// =========================================================
// 0. SYSTEM SAFE (oba NC stop prekidača moraju biti OK)
// =========================================================
bSystemSafe := GVL_IO.DI_Stop_Port AND GVL_IO.DI_Stop_Stbd;

// =========================================================
// 1. POZIV FUNKCIJSKIH BLOKOVA ZA VINČEVE
// =========================================================

// WINCH 1
fbWinch1(
    bIn_SafetyEnable := bSystemSafe,
    bBtn_Phy_Dir1    := GVL_IO.bBtn_Winch1_A,
    bBtn_Phy_Dir2    := GVL_IO.bBtn_Winch1_B,
    stHMI            := stWinch1_HMI,
    bValve_Dir1      => GVL_IO.bValve_Winch1_A,
    bValve_Dir2      => GVL_IO.bValve_Winch1_B
);

// WINCH 2
fbWinch2(
    bIn_SafetyEnable := bSystemSafe,
    bBtn_Phy_Dir1    := GVL_IO.bBtn_Winch2_A,
    bBtn_Phy_Dir2    := GVL_IO.bBtn_Winch2_B,
    stHMI            := stWinch2_HMI,
    bValve_Dir1      => GVL_IO.bValve_Winch2_A,
    bValve_Dir2      => GVL_IO.bValve_Winch2_B
);

// WINCH 3
fbWinch3(
    bIn_SafetyEnable := bSystemSafe,
    bBtn_Phy_Dir1    := GVL_IO.bBtn_Winch3_A,
    bBtn_Phy_Dir2    := GVL_IO.bBtn_Winch3_B,
    stHMI            := stWinch3_HMI,
    bValve_Dir1      => GVL_IO.bValve_Winch3_A,
    bValve_Dir2      => GVL_IO.bValve_Winch3_B
);

// =========================================================
// 2. DETEKCIJA OPTEREĆENJA (Koliko vinčeva radi?)
// =========================================================
iActiveCount := 0;

// Sada gledamo čisti izlaz iz FB-a koji već u sebi ima interlock i logiku!
IF fbWinch1.bReq_Pump THEN iActiveCount := iActiveCount + 1; END_IF
IF fbWinch2.bReq_Pump THEN iActiveCount := iActiveCount + 1; END_IF
IF fbWinch3.bReq_Pump THEN iActiveCount := iActiveCount + 1; END_IF

// Zastavica: Radi li itko?
GVL_IO.bAnyWinchActive := (iActiveCount > 0);

// =========================================================
// 3. UPRAVLJANJE RPM-om MOTORA (BOOST)
// =========================================================
bEngineIsOn := (GVL_IO.fEngineRPM_Scaled > 500.0);

IF GVL_IO.bAnyWinchActive AND bEngineIsOn THEN
    // Formula: Bazni ler + (BrojVinčeva * 200)
    GVL_IO.iRpmReq_Winches := iBaseRpm + (iActiveCount * iRpmPerWinch);
    
    // Sigurnosni limit RPM-a
    IF GVL_IO.iRpmReq_Winches > 2000 THEN 
        GVL_IO.iRpmReq_Winches := 2000; 
    END_IF
ELSE
    // Ako vinčevi ne rade ili motor stoji
    GVL_IO.iRpmReq_Winches := 0; 
END_IF

// =========================================================
// 4. LOGIKA DC PUMPE (BACKUP S OFF-DELAY TIMEMEROM)
// =========================================================

// Ako netko stišće vinč, a glavni motor ne vrti
// TOF (Timer Off) se pali momentalno, a gasi tek 5 sekundi nakon što pustiš tipku
tmrDCPumpOff(
    IN := (GVL_IO.bAnyWinchActive AND NOT bEngineIsOn), 
    PT := T#5S
);

GVL_IO.bDcPump_Start := tmrDCPumpOff.Q;

END_PROGRAM

// ---- POUs/FBs/FB_WinchControl.TcPOU
FUNCTION_BLOCK FB_WinchControl
VAR_INPUT
    (* --- FIZIČKI ULAZI --- *)
	bIn_SafetyEnable : BOOL;
    bBtn_Phy_Dir1    : BOOL; (* Fizička tipka (npr. nožni prekidač Slow) *)
    bBtn_Phy_Dir2    : BOOL; (* Fizička tipka (npr. nožni prekidač Fast) *)
END_VAR
VAR_OUTPUT
    (* --- FIZIČKI IZLAZI --- *)
    bValve_Dir1      : BOOL; 
    bValve_Dir2      : BOOL; 
    bReq_Pump        : BOOL; 
END_VAR
VAR_IN_OUT
    (* --- HMI PODACI --- *)
    stHMI            : ST_UcWinchControl;
END_VAR
VAR
    xCmd_Dir1        : BOOL;
    xCmd_Dir2        : BOOL;
END_VAR

(* ========================================================== *)
(* 1. INPUT MIXER (HMI vs HARDVER)                            *)
(* ========================================================== *)
IF stHMI.bManualEnable THEN
    (* Manual Mode: Slušamo samo HMI *)
    xCmd_Dir1 := stHMI.bBtn_Dir1;
    xCmd_Dir2 := stHMI.bBtn_Dir2;
ELSE
    (* Local Mode: Slušamo samo fizičke tipke *)
    xCmd_Dir1 := bBtn_Phy_Dir1;
    xCmd_Dir2 := bBtn_Phy_Dir2;
END_IF;

(* ========================================================== *)
(* 2. LOGIKA VITLA (Interlock + Pumpa)                        *)
(* ========================================================== *)
IF bIn_SafetyEnable AND NOT stHMI.bDisable THEN
    
    // Interlock: Ne može obje brzine/smjera odjednom
    IF xCmd_Dir1 AND xCmd_Dir2 THEN
        bValve_Dir1 := FALSE;
        bValve_Dir2 := FALSE;
        bReq_Pump   := FALSE;

    // Smjer 1 (npr. Slow / In)
    ELSIF xCmd_Dir1 THEN
        bValve_Dir1 := TRUE;
        bValve_Dir2 := FALSE;
        bReq_Pump   := TRUE; (* PUMPA ON *)

    // Smjer 2 (npr. Fast / Out)
    ELSIF xCmd_Dir2 THEN
        bValve_Dir1 := FALSE;
        bValve_Dir2 := TRUE;
        bReq_Pump   := TRUE; (* PUMPA ON *)
    
    // Mirovanje
    ELSE
        bValve_Dir1 := FALSE;
        bValve_Dir2 := FALSE;
        bReq_Pump   := FALSE;
    END_IF

ELSE
    // SAFETY STOP
    bValve_Dir1 := FALSE;
    bValve_Dir2 := FALSE;
    bReq_Pump   := FALSE;
END_IF

(* ========================================================== *)
(* 3. HMI FEEDBACK (Update strukture)                         *)
(* ========================================================== *)
stHMI.bValve_Dir1     := bValve_Dir1;
stHMI.bValve_Dir2     := bValve_Dir2;
stHMI.bReq_Pump       := bReq_Pump;

stHMI.bSts_SystemSafe := bIn_SafetyEnable AND NOT stHMI.bDisable;
stHMI.bSts_ManualEn   := stHMI.bManualEnable;

END_FUNCTION_BLOCK

// ---- POUs/Sim/PRG_SimDoors.TcPOU
PROGRAM PRG_SimDoors
VAR
    (* Parametri za VRATA *)
    fRiseSpeed   : REAL := 0.04; 
    fDropSpeed   : REAL := 0.001; 
    fTankSpeed   : REAL := 2.0;  
    
    (* Tajmeri za simulaciju kretanja VENTILA *)
    tonP1, tonP2, tonP3 : TON;
    tonS1, tonS2, tonS3 : TON;
    tonTunel           : TON;
    
    tValveTime : TIME := T#1.5S; (* Brže od 3s timeouta u FB-u! *)
    bSimActive : BOOL := TRUE;
	
	// Timer koji simulira koliko dugo ima vode u cijevima nakon paljenja pumpe
	tmrVodaTrajanje : TON;
    tVrijemeRada    : TIME := T#10S; // Koliko dugo ima vode u tanku
    bTankPrazan     : BOOL;         // Zasun koji sprječava titranjeEND_VAR
END_VAR

// -----------------------------------------------------------
// 0. GLAVNI PREKIDAČ SIMULATORA
// -----------------------------------------------------------
IF NOT bSimActive THEN
    RETURN;
END_IF

// -----------------------------------------------------------
// 1. SIMULACIJA VRATA (FWD & AFT)
// -----------------------------------------------------------

// --- FWD VRATA ---
IF GVL_IO.DO_DoorFwd_Open THEN
    GVL_IO.fPressure_FWD_A := GVL_IO.fPressure_FWD_A + fRiseSpeed;
    GVL_IO.fPressure_FWD_B := GVL_IO.fPressure_FWD_B - fTankSpeed;
ELSIF GVL_IO.DO_DoorFwd_Close THEN
    GVL_IO.fPressure_FWD_B := GVL_IO.fPressure_FWD_B + fRiseSpeed;
    GVL_IO.fPressure_FWD_A := GVL_IO.fPressure_FWD_A - fTankSpeed;
ELSE
    GVL_IO.fPressure_FWD_A := GVL_IO.fPressure_FWD_A - fDropSpeed;
    GVL_IO.fPressure_FWD_B := GVL_IO.fPressure_FWD_B - fDropSpeed;
END_IF

// --- AFT VRATA ---
IF GVL_IO.DO_DoorAft_Open THEN
    GVL_IO.fPressure_AFT_A := GVL_IO.fPressure_AFT_A + fRiseSpeed;
    GVL_IO.fPressure_AFT_B := GVL_IO.fPressure_AFT_B - fTankSpeed;
ELSIF GVL_IO.DO_DoorAft_Close THEN
    GVL_IO.fPressure_AFT_B := GVL_IO.fPressure_AFT_B + fRiseSpeed;
    GVL_IO.fPressure_AFT_A := GVL_IO.fPressure_AFT_A - fTankSpeed;
ELSE
    GVL_IO.fPressure_AFT_A := GVL_IO.fPressure_AFT_A - fDropSpeed;
    GVL_IO.fPressure_AFT_B := GVL_IO.fPressure_AFT_B - fDropSpeed;
END_IF

// Ograničenja tlaka (da ne ide u minus ili beskonačno)
GVL_IO.fPressure_FWD_A := LIMIT(0.0, GVL_IO.fPressure_FWD_A, 150.0);
GVL_IO.fPressure_FWD_B := LIMIT(0.0, GVL_IO.fPressure_FWD_B, 150.0);
GVL_IO.fPressure_AFT_A := LIMIT(0.0, GVL_IO.fPressure_AFT_A, 150.0);
GVL_IO.fPressure_AFT_B := LIMIT(0.0, GVL_IO.fPressure_AFT_B, 150.0);

// -----------------------------------------------------------
// 2. SIMULACIJA BALAST VENTILA (Feedback)
// -----------------------------------------------------------

// PORT 1
tonP1(IN := GVL_IO.DO_BAL_P1, PT := tValveTime);
IF GVL_IO.DO_BAL_P1 THEN
    GVL_IO.DI_BAL_P1_OPEN_FB  := tonP1.Q;
    GVL_IO.DI_BAL_P1_CLOSE_FB := FALSE;
ELSE
    GVL_IO.DI_BAL_P1_OPEN_FB  := FALSE;
    GVL_IO.DI_BAL_P1_CLOSE_FB := TRUE;
END_IF

// PORT 2
tonP2(IN := GVL_IO.DO_BAL_P2, PT := tValveTime);
IF GVL_IO.DO_BAL_P2 THEN
    GVL_IO.DI_BAL_P2_OPEN_FB  := tonP2.Q;
    GVL_IO.DI_BAL_P2_CLOSE_FB := FALSE;
ELSE
    GVL_IO.DI_BAL_P2_OPEN_FB  := FALSE;
    GVL_IO.DI_BAL_P2_CLOSE_FB := TRUE;
END_IF

// PORT 3
tonP3(IN := GVL_IO.DO_BAL_P3, PT := tValveTime);
IF GVL_IO.DO_BAL_P3 THEN
    GVL_IO.DI_BAL_P3_OPEN_FB  := tonP3.Q;
    GVL_IO.DI_BAL_P3_CLOSE_FB := FALSE;
ELSE
    GVL_IO.DI_BAL_P3_OPEN_FB  := FALSE;
    GVL_IO.DI_BAL_P3_CLOSE_FB := TRUE;
END_IF

// STBD 1
tonS1(IN := GVL_IO.DO_BAL_S1, PT := tValveTime);
IF GVL_IO.DO_BAL_S1 THEN
    GVL_IO.DI_BAL_S1_OPEN_FB  := tonS1.Q;
    GVL_IO.DI_BAL_S1_CLOSE_FB := FALSE;
ELSE
    GVL_IO.DI_BAL_S1_OPEN_FB  := FALSE;
    GVL_IO.DI_BAL_S1_CLOSE_FB := TRUE;
END_IF

// STBD 2
tonS2(IN := GVL_IO.DO_BAL_S2, PT := tValveTime);
IF GVL_IO.DO_BAL_S2 THEN
    GVL_IO.DI_BAL_S2_OPEN_FB  := tonS2.Q;
    GVL_IO.DI_BAL_S2_CLOSE_FB := FALSE;
ELSE
    GVL_IO.DI_BAL_S2_OPEN_FB  := FALSE;
    GVL_IO.DI_BAL_S2_CLOSE_FB := TRUE;
END_IF

// STBD 3
tonS3(IN := GVL_IO.DO_BAL_S3, PT := tValveTime);
IF GVL_IO.DO_BAL_S3 THEN
    GVL_IO.DI_BAL_S3_OPEN_FB  := tonS3.Q;
    GVL_IO.DI_BAL_S3_CLOSE_FB := FALSE;
ELSE
    GVL_IO.DI_BAL_S3_OPEN_FB  := FALSE;
    GVL_IO.DI_BAL_S3_CLOSE_FB := TRUE;
END_IF

// -----------------------------------------------------------
// 3. SIMULACIJA TUNEL PUMP VENTILA
// -----------------------------------------------------------
tonTunel(IN := GVL_IO.DO_TUNEL_VALVE, PT := tValveTime);
IF GVL_IO.DO_TUNEL_VALVE THEN
    GVL_IO.DI_TUNEL_OPEN_FB  := tonTunel.Q;
    GVL_IO.DI_TUNEL_CLOSE_FB := FALSE;
ELSE
    GVL_IO.DI_TUNEL_OPEN_FB  := FALSE;
    GVL_IO.DI_TUNEL_CLOSE_FB := TRUE;
END_IF

// ==========================================================
// 4. SIMULACIJA SONDI S TIMEROM (NESTANAK VODE)
// ==========================================================

// --- SIMULACIJA NESTANKA VODE ---
// Timer mjeri koliko dugo pumpa (Clutch) vrti
tmrVodaTrajanje(IN := GVL_IO.DO_TunelClutch, PT := tVrijemeRada);

// Kad timer odradi, "ispraznili" smo tank
IF tmrVodaTrajanje.Q THEN
    bTankPrazan := TRUE; 
END_IF

// Resetiramo tank tek kad se ugasi komanda pumpe (da možemo opet testirati)
IF NOT GVL_HMI.bCmdRun_TunelPump THEN
    bTankPrazan := FALSE;
END_IF

// --- LOGIKA SONDI ---
IF GVL_IO.DO_SondePower THEN
    // Port Sonda: ima struje, ventil je na Portu I tank NIJE prazan
    GVL_IO.DI_Sonda_Port := GVL_IO.DI_TUNEL_OPEN_FB AND NOT bTankPrazan;
    
    // Stbd Sonda: ima struje, ventil je na Stbd I tank NIJE prazan
    GVL_IO.DI_Sonda_Stbd := GVL_IO.DI_TUNEL_CLOSE_FB AND NOT bTankPrazan;
ELSE
    GVL_IO.DI_Sonda_Port := FALSE;
    GVL_IO.DI_Sonda_Stbd := FALSE;
END_IF

END_PROGRAM

// ---- POUs/PRG_HmiLeds.TcPOU
PROGRAM PRG_HmiLeds
VAR
END_VAR


// ============================================================
// HMI LED STATUSI
// Cyan=Otvoren, Green=Zatvoren, Orange(Yellow)=Putuje, Red=Greška
// ============================================================

// --- MOTOR ---
GVL_HMI.bLed_Engine_Green := GVL_ENGINE.bEngineRunning;

// --- PUMPA ---
GVL_HMI.bLed_Pump_Cyan := GVL_HMI.bCmdRun_TunelPump;
GVL_HMI.bLed_Pump_Red  := FALSE;

// --- PORT VENTILI ---
// P1
IF GVL_HMI.bAlarm_P1 THEN
    GVL_HMI.bLed_P1_Red := TRUE;  GVL_HMI.bLed_P1_Cyan := FALSE; GVL_HMI.bLed_P1_Yellow := FALSE; GVL_HMI.bLed_P1_Green := FALSE;
ELSIF GVL_HMI.eState_P1 = E_ValveState.VALVE_OPEN THEN
    GVL_HMI.bLed_P1_Red := FALSE; GVL_HMI.bLed_P1_Cyan := TRUE;  GVL_HMI.bLed_P1_Yellow := FALSE; GVL_HMI.bLed_P1_Green := FALSE;
ELSIF GVL_HMI.eState_P1 = E_ValveState.VALVE_UNKNOWN THEN
    GVL_HMI.bLed_P1_Red := FALSE; GVL_HMI.bLed_P1_Cyan := FALSE; GVL_HMI.bLed_P1_Yellow := TRUE;  GVL_HMI.bLed_P1_Green := FALSE;
ELSE // VALVE_CLOSED
    GVL_HMI.bLed_P1_Red := FALSE; GVL_HMI.bLed_P1_Cyan := FALSE; GVL_HMI.bLed_P1_Yellow := FALSE; GVL_HMI.bLed_P1_Green := TRUE;
END_IF

// P2
IF GVL_HMI.bAlarm_P2 THEN
    GVL_HMI.bLed_P2_Red := TRUE;  GVL_HMI.bLed_P2_Cyan := FALSE; GVL_HMI.bLed_P2_Yellow := FALSE; GVL_HMI.bLed_P2_Green := FALSE;
ELSIF GVL_HMI.eState_P2 = E_ValveState.VALVE_OPEN THEN
    GVL_HMI.bLed_P2_Red := FALSE; GVL_HMI.bLed_P2_Cyan := TRUE;  GVL_HMI.bLed_P2_Yellow := FALSE; GVL_HMI.bLed_P2_Green := FALSE;
ELSIF GVL_HMI.eState_P2 = E_ValveState.VALVE_UNKNOWN THEN
    GVL_HMI.bLed_P2_Red := FALSE; GVL_HMI.bLed_P2_Cyan := FALSE; GVL_HMI.bLed_P2_Yellow := TRUE;  GVL_HMI.bLed_P2_Green := FALSE;
ELSE
    GVL_HMI.bLed_P2_Red := FALSE; GVL_HMI.bLed_P2_Cyan := FALSE; GVL_HMI.bLed_P2_Yellow := FALSE; GVL_HMI.bLed_P2_Green := TRUE;
END_IF

// P3
IF GVL_HMI.bAlarm_P3 THEN
    GVL_HMI.bLed_P3_Red := TRUE;  GVL_HMI.bLed_P3_Cyan := FALSE; GVL_HMI.bLed_P3_Yellow := FALSE; GVL_HMI.bLed_P3_Green := FALSE;
ELSIF GVL_HMI.eState_P3 = E_ValveState.VALVE_OPEN THEN
    GVL_HMI.bLed_P3_Red := FALSE; GVL_HMI.bLed_P3_Cyan := TRUE;  GVL_HMI.bLed_P3_Yellow := FALSE; GVL_HMI.bLed_P3_Green := FALSE;
ELSIF GVL_HMI.eState_P3 = E_ValveState.VALVE_UNKNOWN THEN
    GVL_HMI.bLed_P3_Red := FALSE; GVL_HMI.bLed_P3_Cyan := FALSE; GVL_HMI.bLed_P3_Yellow := TRUE;  GVL_HMI.bLed_P3_Green := FALSE;
ELSE
    GVL_HMI.bLed_P3_Red := FALSE; GVL_HMI.bLed_P3_Cyan := FALSE; GVL_HMI.bLed_P3_Yellow := FALSE; GVL_HMI.bLed_P3_Green := TRUE;
END_IF

// --- STBD VENTILI ---
// S1
IF GVL_HMI.bAlarm_S1 THEN
    GVL_HMI.bLed_S1_Red := TRUE;  GVL_HMI.bLed_S1_Cyan := FALSE; GVL_HMI.bLed_S1_Yellow := FALSE; GVL_HMI.bLed_S1_Green := FALSE;
ELSIF GVL_HMI.eState_S1 = E_ValveState.VALVE_OPEN THEN
    GVL_HMI.bLed_S1_Red := FALSE; GVL_HMI.bLed_S1_Cyan := TRUE;  GVL_HMI.bLed_S1_Yellow := FALSE; GVL_HMI.bLed_S1_Green := FALSE;
ELSIF GVL_HMI.eState_S1 = E_ValveState.VALVE_UNKNOWN THEN
    GVL_HMI.bLed_S1_Red := FALSE; GVL_HMI.bLed_S1_Cyan := FALSE; GVL_HMI.bLed_S1_Yellow := TRUE;  GVL_HMI.bLed_S1_Green := FALSE;
ELSE
    GVL_HMI.bLed_S1_Red := FALSE; GVL_HMI.bLed_S1_Cyan := FALSE; GVL_HMI.bLed_S1_Yellow := FALSE; GVL_HMI.bLed_S1_Green := TRUE;
END_IF

// S2
IF GVL_HMI.bAlarm_S2 THEN
    GVL_HMI.bLed_S2_Red := TRUE;  GVL_HMI.bLed_S2_Cyan := FALSE; GVL_HMI.bLed_S2_Yellow := FALSE; GVL_HMI.bLed_S2_Green := FALSE;
ELSIF GVL_HMI.eState_S2 = E_ValveState.VALVE_OPEN THEN
    GVL_HMI.bLed_S2_Red := FALSE; GVL_HMI.bLed_S2_Cyan := TRUE;  GVL_HMI.bLed_S2_Yellow := FALSE; GVL_HMI.bLed_S2_Green := FALSE;
ELSIF GVL_HMI.eState_S2 = E_ValveState.VALVE_UNKNOWN THEN
    GVL_HMI.bLed_S2_Red := FALSE; GVL_HMI.bLed_S2_Cyan := FALSE; GVL_HMI.bLed_S2_Yellow := TRUE;  GVL_HMI.bLed_S2_Green := FALSE;
ELSE
    GVL_HMI.bLed_S2_Red := FALSE; GVL_HMI.bLed_S2_Cyan := FALSE; GVL_HMI.bLed_S2_Yellow := FALSE; GVL_HMI.bLed_S2_Green := TRUE;
END_IF

// S3
IF GVL_HMI.bAlarm_S3 THEN
    GVL_HMI.bLed_S3_Red := TRUE;  GVL_HMI.bLed_S3_Cyan := FALSE; GVL_HMI.bLed_S3_Yellow := FALSE; GVL_HMI.bLed_S3_Green := FALSE;
ELSIF GVL_HMI.eState_S3 = E_ValveState.VALVE_OPEN THEN
    GVL_HMI.bLed_S3_Red := FALSE; GVL_HMI.bLed_S3_Cyan := TRUE;  GVL_HMI.bLed_S3_Yellow := FALSE; GVL_HMI.bLed_S3_Green := FALSE;
ELSIF GVL_HMI.eState_S3 = E_ValveState.VALVE_UNKNOWN THEN
    GVL_HMI.bLed_S3_Red := FALSE; GVL_HMI.bLed_S3_Cyan := FALSE; GVL_HMI.bLed_S3_Yellow := TRUE;  GVL_HMI.bLed_S3_Green := FALSE;
ELSE
    GVL_HMI.bLed_S3_Red := FALSE; GVL_HMI.bLed_S3_Cyan := FALSE; GVL_HMI.bLed_S3_Yellow := FALSE; GVL_HMI.bLed_S3_Green := TRUE;
END_IF

// --- TUNEL VENTIL ---
IF GVL_HMI.bAlarm_Tunel THEN
    GVL_HMI.bLed_Tunel_Red := TRUE;  GVL_HMI.bLed_Tunel_Cyan := FALSE; GVL_HMI.bLed_Tunel_Yellow := FALSE; GVL_HMI.bLed_Tunel_Green := FALSE;
ELSIF GVL_HMI.eState_Tunel = E_ValveState.VALVE_OPEN THEN
    GVL_HMI.bLed_Tunel_Red := FALSE; GVL_HMI.bLed_Tunel_Cyan := TRUE;  GVL_HMI.bLed_Tunel_Yellow := FALSE; GVL_HMI.bLed_Tunel_Green := FALSE;
ELSIF GVL_HMI.eState_Tunel = E_ValveState.VALVE_UNKNOWN THEN
    GVL_HMI.bLed_Tunel_Red := FALSE; GVL_HMI.bLed_Tunel_Cyan := FALSE; GVL_HMI.bLed_Tunel_Yellow := TRUE;  GVL_HMI.bLed_Tunel_Green := FALSE;
ELSE
    GVL_HMI.bLed_Tunel_Red := FALSE; GVL_HMI.bLed_Tunel_Cyan := FALSE; GVL_HMI.bLed_Tunel_Yellow := FALSE; GVL_HMI.bLed_Tunel_Green := TRUE;
END_IF

// --- VRATA FWD ---
IF GVL_HMI.bAlarm_DoorFwd THEN
    GVL_HMI.bLed_DoorFwd_Red := TRUE;  GVL_HMI.bLed_DoorFwd_Cyan := FALSE; GVL_HMI.bLed_DoorFwd_Yellow := FALSE; GVL_HMI.bLed_DoorFwd_Green := FALSE;
ELSIF GVL_HMI.eState_DoorFwd = 1 THEN // OPEN
    GVL_HMI.bLed_DoorFwd_Red := FALSE; GVL_HMI.bLed_DoorFwd_Cyan := TRUE;  GVL_HMI.bLed_DoorFwd_Yellow := FALSE; GVL_HMI.bLed_DoorFwd_Green := FALSE;
ELSIF GVL_HMI.eState_DoorFwd = 0 THEN // PUTUJE
    GVL_HMI.bLed_DoorFwd_Red := FALSE; GVL_HMI.bLed_DoorFwd_Cyan := FALSE; GVL_HMI.bLed_DoorFwd_Yellow := TRUE;  GVL_HMI.bLed_DoorFwd_Green := FALSE;
ELSE // CLOSED
    GVL_HMI.bLed_DoorFwd_Red := FALSE; GVL_HMI.bLed_DoorFwd_Cyan := FALSE; GVL_HMI.bLed_DoorFwd_Yellow := FALSE; GVL_HMI.bLed_DoorFwd_Green := TRUE;
END_IF

// --- VRATA AFT ---
IF GVL_HMI.bAlarm_DoorAft THEN
    GVL_HMI.bLed_DoorAft_Red := TRUE;  GVL_HMI.bLed_DoorAft_Cyan := FALSE; GVL_HMI.bLed_DoorAft_Yellow := FALSE; GVL_HMI.bLed_DoorAft_Green := FALSE;
ELSIF GVL_HMI.eState_DoorAft = 1 THEN // OPEN
    GVL_HMI.bLed_DoorAft_Red := FALSE; GVL_HMI.bLed_DoorAft_Cyan := TRUE;  GVL_HMI.bLed_DoorAft_Yellow := FALSE; GVL_HMI.bLed_DoorAft_Green := FALSE;
ELSIF GVL_HMI.eState_DoorAft = 0 THEN // PUTUJE
    GVL_HMI.bLed_DoorAft_Red := FALSE; GVL_HMI.bLed_DoorAft_Cyan := FALSE; GVL_HMI.bLed_DoorAft_Yellow := TRUE;  GVL_HMI.bLed_DoorAft_Green := FALSE;
ELSE // CLOSED
    GVL_HMI.bLed_DoorAft_Red := FALSE; GVL_HMI.bLed_DoorAft_Cyan := FALSE; GVL_HMI.bLed_DoorAft_Yellow := FALSE; GVL_HMI.bLed_DoorAft_Green := TRUE;
END_IF

END_PROGRAM

// ---- POUs/DirectMotorControl.TcPOU
PROGRAM DirectMotorControl
VAR
	bHMI_RESET: BOOL;	// reset gresaka
 
	bMotorOn: BOOL;
	rVelocitySetpoint: LREAL;
	rPotFeedback_V: REAL;
	rPotFeedback_Radno_Perc: LREAL;
	rRadno_Min_Pos: LREAL;	// Radni limit 0%
	rRadno_Max_Pos: REAL;	// Radni limit 100%
	
   // Realni Potenciometar - u RAW vrijednosti
    cPotMin: REAL := 0.55;             // kΩ ili V
    cPotMax: REAL := 7.16;             // kΩ ili V
	rLinearPosition: LREAL;	// realna pozicija max hoda od 81mm

	rLinearPosition_LimMin: LREAL;	// Limit iskljucenja
	rLinearPosition_LimMAx: LREAL;	// Limit iskljucenja
	
	// Parametri regulacije (NOVO)
    rSetpoint: REAL := 50.0;      // Željena pozicija 0-100%
    rMinVelocity: REAL := 10.0;     // Min brzina za start %
    rMaxVelocity: REAL := 100.0;   // Max brzina %
    rDeadband: REAL := 1.0;        // Deadband ±1%
    rKp: REAL := 10;              // P pojačanje
    
    // Procesne varijable (NOVO)
    rError: REAL;	// greska slijeđenja
    rVelocityCmd: REAL;
    bInDeadband: BOOL;	// Unutar pozicije
	
   // NOVO - Rampa varijable
    rSetpointTarget: REAL := 50.0;    // Ciljna pozicija
    rRampRate: REAL := 50.0;          // Brzina rampe [%/s]
	
   // NOVO - Računanje brzine
    rActualVelocity: REAL;        // Stvarna brzina [%/s]
    rActualVelocityRPM: REAL;     // Stvarna brzina [RPM]
    rLastPosition: LREAL;          // Prethodna pozicija
    rDeltaPosition: LREAL;         // Promjena pozicije
    fbVelocityTimer: TON;         // Timer za uzorkovanje
    tSampleTime: TIME := T#50MS;  // Vrijeme uzorkovanja
    
    // Filter za brzinu (opciono)
    rVelocityFiltered: REAL;
    rFilterConst: REAL := 0.3;    // Filter konstanta (0.1-0.5)

	rMotorVoltage: LREAL;
	rMotorCurrent: LREAL;
	Tgen1: TON;
	bTick: BOOL;
	TP1: TP;
	bTakt: BOOL;
	rSetpointTarget_Min: REAL:=0.0;
	rSetpointTarget_Max: REAL:=100.0;
	
	bSetVelOverPoz: BOOL;
	bSetVelOverNeg: BOOL;
	
	R_Tgen1: R_TRIG;

	Kn: REAL;
END_VAR

// Test postavke za reverziranje 0..100%
(*
Tgen1(IN:=NOT bTick , PT:=T#5S , Q=>bTick , ET=> );
TP1(IN:=bTick , PT:=Tgen1.PT/2 , Q=>bTakt , ET=> );
*)
Tgen1(IN:=bInDeadband , PT:=T#2S , Q=>bTick , ET=> );
R_Tgen1(CLK:=Tgen1.Q , Q=>bTick );
IF bTick THEN
	bTakt:=NOT bTakt;
END_IF

// MODIFICIRANO - postavljamo target umjesto direktnog setpointa
IF bTakt THEN
    rSetpointTarget := rSetpointTarget_Min;
ELSE
    rSetpointTarget := rSetpointTarget_Max;
END_IF

// NOVO - Rampiranje setpointa
IF rSetpoint < rSetpointTarget - 0.1 THEN
    // Rampiranje gore
    rSetpoint := rSetpoint + rRampRate * 0.01; // 0.01 = 10ms ciklus
    IF rSetpoint > rSetpointTarget THEN
        rSetpoint := rSetpointTarget;
    END_IF
ELSIF rSetpoint > rSetpointTarget + 0.1 THEN
    // Rampiranje dolje  
    rSetpoint := rSetpoint - rRampRate * 0.01;
    IF rSetpoint < rSetpointTarget THEN
        rSetpoint := rSetpointTarget;
    END_IF
END_IF


// Skaliranje 1 okretajng pot pozicije.
rPotFeedback_V:=10.0*iwPotFeedback/32767;	//napon na ulazu u EL3002
// pozicija pomaka = 81mm
rLinearPosition:=81.0*(rPotFeedback_V-cPotMin)/(cPotMax-cPotMin);
// Sigurnosni limiti + / - 
rLinearPosition_LimMin:=5.0;	// Safe limit negativan
rLinearPosition_LimMAx:=75.0;	// Safe limit pozitivan

// Sigurnosni limiti - iskljucuju Motor
IF (rLinearPosition < rLinearPosition_LimMin) OR  (rLinearPosition > rLinearPosition_LimMAx) THEN
	bMotorOn:=FALSE;
END_IF

// Radno podrucje pomaka 0..100% = MORA BITI UNUTAR SIGURNOSNIH LIMITA
rRadno_Min_Pos:=10.0;
rRadno_Max_Pos:=70.0;
rPotFeedback_Radno_Perc:= 100*(rLinearPosition-rRadno_Min_Pos)/(rRadno_Max_Pos-rRadno_Min_Pos);

// Open-loop kontrola
// Setpoint 0..100% = 0.....
// Limit za pretvorbu u integer 
// greska ako je veće od 32766 i manje od - 32766

// Kn ke multiplikator za setpoint u granicama -32000 .. 32000 / 0.100%
Kn:=320; // ako ide do napona napajanja 12V onda na 100% steka
// reset iz HMI
// bReset := FALSE;
IF bHMI_RESET THEN
	bSetVelOverPoz:=FALSE;
	bSetVelOverNeg:=FALSE;
    bReset := TRUE;
END_IF

IF NOT bError THEN
	bReset := FALSE;
END_IF


IF (rVelocitySetpoint*Kn > 32766) THEN
	bSetVelOverPoz:=TRUE;
END_IF
IF (rVelocitySetpoint*Kn < -32766) THEN
	bSetVelOverNeg:=TRUE;
END_IF
IF bSetVelOverPoz OR bSetVelOverNeg THEN
	bMotorOn:=FALSE;
ELSE
	nVelocitySetpoint:=LREAL_TO_INT(rVelocitySetpoint*Kn);
END_IF

// Dodano
// NOVO - POZICIJSKA REGULACIJA
IF bMotorOn THEN
    // Računaj grešku pozicije
    rError := rSetpoint - rPotFeedback_Radno_Perc;
    
    // Provjeri deadband
    bInDeadband := ABS(rError) <= rDeadband;
    
    IF NOT bInDeadband THEN
        // P regulator
        rVelocityCmd := rError * rKp;
        
        // Ograniči na max brzinu
        rVelocityCmd := LIMIT(-rMaxVelocity, rVelocityCmd, rMaxVelocity);
        
        // Primjeni minimalnu brzinu
        IF (ABS(rVelocityCmd) > 0.1) AND (ABS(rVelocityCmd) < rMinVelocity) THEN
            IF rVelocityCmd > 0 THEN
                rVelocityCmd := rMinVelocity;
            ELSE
                rVelocityCmd := -rMinVelocity;
            END_IF
        END_IF
    ELSE
        // Unutar deadband - zaustavi
        rVelocityCmd := 0.0;
    END_IF
    
    // Postavi brzinu
    rVelocitySetpoint := rVelocityCmd;
ELSE
    rVelocitySetpoint := 0.0;
END_IF

// Računanje brzine iz promjene pozicije

// Timer za periodičko računanje brzine
fbVelocityTimer(IN:= NOT fbVelocityTimer.Q, PT:= tSampleTime);

// Računaj brzinu kada timer istekne
IF fbVelocityTimer.Q THEN
    // Promjena pozicije u %
    rDeltaPosition := rLinearPosition - rLastPosition;
    
    // Brzina u mm/s !!!! NAVOJ IMA MULTIPLIKATOR X2
    rActualVelocity := rDeltaPosition / 0.05 / 2 ; // 50ms = 0.05s
    
    // Spremi trenutnu poziciju
    rLastPosition := rLinearPosition;
    
    // Filter brzine (PT1)
    rVelocityFiltered := rVelocityFiltered * (1.0 - rFilterConst) + 
                        rActualVelocity * rFilterConst;
END_IF

// Preračun u druge jedinice
// 81mm =  171.3 okr Motora
// RPM motora
rActualVelocityRPM := 60*171.3*rActualVelocity/81 ;


// =======================  DIVER PREMA TERMINALU

// driver prema EL7342
IF bMotorOn THEN
    bEnable := TRUE;
    bReduceTorque := FALSE;  // Puna snaga
 ELSE
    bEnable := FALSE;
    bReduceTorque := FALSE;
    nVelocitySetpoint := 0;
END_IF

(*
IF bMotorOn THEN
    nControlWord := 16#000F;
ELSE
    nControlWord := 16#0006;
    nVelocitySetpoint := 0;
END_IF
*)

rMotorVoltage:=(UINT_TO_INT(nMotorVoltage))/1000.0;
rMotorCurrent:=(UINT_TO_INT(nMotorCurrent))/1000.0;

END_PROGRAM

// ---- POUs/PRG_Sequence.TcPOU
PROGRAM PRG_Sequence
VAR
    eTargetMode  : E_SystemMode := 0;
    bTurbineSafe : BOOL;
    
    (* Nova varijabla: Netko treba vodu *)
    bWaterRequest : BOOL; 
	
	(* Triggeri za Tipku 4 s obje tipkovnice *)
    rtMode_ID10   : R_TRIG;
    rtMode_ID11   : R_TRIG;
END_VAR

// =========================================================
// 1. OBRADA ZAHTJEVA ZA MOD (Tipka 4)
// =========================================================

// Sigurnost: Ne mijenjaj mod ako turbina vrti prebrzo
bTurbineSafe := (GVL_IO.fEngineRPM_Scaled < 900.0); 

rtMode_ID10(CLK := GVL_CAN.ID10_Status[4]);
rtMode_ID11(CLK := GVL_CAN.ID11_Status[4]);

// Ako je sigurno, kružimo kroz modove pritiskom na Tipku 4
IF bTurbineSafe AND (rtMode_ID10.Q OR rtMode_ID11.Q) THEN
    CASE eTargetMode OF
        E_SystemMode.MODE_IDLE:  
            eTargetMode := E_SystemMode.MODE_DRIVE; // Prebaci na Drive (Zeleno)
            
        E_SystemMode.MODE_DRIVE: 
            eTargetMode := E_SystemMode.MODE_SAIL;  // Prebaci na Sail (Plavo)
            
        E_SystemMode.MODE_SAIL:  
            eTargetMode := E_SystemMode.MODE_IDLE;  // Vrati na Idle (Off)
    END_CASE
END_IF

// Zadržavamo i tvoje HMI zahtjeve kao override (ako stisneš na ekranu)
IF bTurbineSafe THEN
    IF GVL_HMI.bReq_Stop THEN eTargetMode := 0;
    ELSIF GVL_HMI.bReq_ModeDrive THEN eTargetMode := 1;
    ELSIF GVL_HMI.bReq_ModeSail  THEN eTargetMode := 2;
    END_IF
END_IF

// =========================================================
// 2. DETEKCIJA ZAHTJEVA ZA VODOM (Ostaje isto)
// =========================================================
bWaterRequest := GVL_HMI.bCmdOpen_P1 OR GVL_HMI.bCmdOpen_P2 OR GVL_HMI.bCmdOpen_P3 OR
                 GVL_HMI.bCmdOpen_S1 OR GVL_HMI.bCmdOpen_S2 OR GVL_HMI.bCmdOpen_S3;

// =========================================================
// 3. UPRAVLJANJE VRATIMA PREMA MODU (Tvoj CASE blok)
// =========================================================
CASE eTargetMode OF
    0:  // MODE_IDLE
        GVL_HMI.bCmdDoorFwd_Open := FALSE; GVL_HMI.bCmdDoorFwd_Close := TRUE;
        GVL_HMI.bCmdDoorAft_Open := FALSE; GVL_HMI.bCmdDoorAft_Close := TRUE;
        GVL_HMI.bSequenceReady := FALSE;

    1:  // MODE_DRIVE (Oba vrata otvorena)
        GVL_HMI.bCmdDoorFwd_Open := TRUE; GVL_HMI.bCmdDoorFwd_Close := FALSE;
        GVL_HMI.bCmdDoorAft_Open := TRUE; GVL_HMI.bCmdDoorAft_Close := FALSE;
        GVL_HMI.bSequenceReady := (GVL_HMI.eState_DoorFwd = 1) AND (GVL_HMI.eState_DoorAft = 1);

    2:  // MODE_SAIL (Zadnja zatvorena, prednja po potrebi)
        GVL_HMI.bCmdDoorAft_Open := FALSE; GVL_HMI.bCmdDoorAft_Close := TRUE;
        IF bWaterRequest THEN
            GVL_HMI.bCmdDoorFwd_Open := TRUE; GVL_HMI.bCmdDoorFwd_Close := FALSE;
        ELSE
            GVL_HMI.bCmdDoorFwd_Open := FALSE; GVL_HMI.bCmdDoorFwd_Close := TRUE;
        END_IF
        GVL_HMI.bSequenceReady := (GVL_HMI.eState_DoorAft = 2);
END_CASE

// Update statusa za HMI i VIZUALIZACIJA TIPKE 4
GVL_HMI.eActiveMode := eTargetMode;

CASE eTargetMode OF
    E_SystemMode.MODE_IDLE:
        GVL_CAN.ID10_Config[4].Boja := GVL_CAN.ID11_Config[4].Boja := 0; // OFF
    E_SystemMode.MODE_DRIVE:
        GVL_CAN.ID10_Config[4].Boja := GVL_CAN.ID11_Config[4].Boja := 2; // ZELENO
    E_SystemMode.MODE_SAIL:
        GVL_CAN.ID10_Config[4].Boja := GVL_CAN.ID11_Config[4].Boja := 3; // PLAVO
END_CASE

END_PROGRAM

// ---- POUs/PRG_StationManager.TcPOU
PROGRAM PRG_StationManager
VAR
	fbStation : FB_StationManager;
END_VAR

fbStation(
    bBtn1 := GVL_IO.bBtn_Sel_St1,
    bBtn2 := GVL_IO.bBtn_Sel_St2,
    iPot1 := GVL_IO.iLever_St1_Raw,
    iPot2 := GVL_IO.iLever_St2_Raw,
    bActiveSt1 => GVL_IO.bLed_Sel_St1,
    bActiveSt2 => GVL_IO.bLed_Sel_St2,
    bBuzzerOut => GVL_IO.bBuzzer,
    iSelectedPot => GVL_IO.iActiveLever_Raw
);

END_PROGRAM

// ---- POUs/PRG_Can.TcPOU
PROGRAM PRG_CAN
VAR
    i           : INT;
    byMaskUSINT : USINT;
    byMaskUINT  : UINT;
    bInitDone   : BOOL := FALSE;
END_VAR

END_PROGRAM

// ---- GlobalTextList.TcGTLO
TEXTLIST GlobalTextList
  205 = ' %Pozicija %.1f '
  801 = '%'
  56 = '% Greska Poz %.1f '
  303 = '% Pozicija %.1f '
  417 = '% Set Poz %.1f '
  331 = '%f'
  794 = '%Greska Poz %.1f '
  685 = 'DI 1'
  587 = 'DI 2'
  904 = 'Enable'
  637 = 'Error'
  435 = 'Error Pos'
  862 = 'ggg'
  618 = 'Greska Poz %.1f '
  68 = 'Lim.Max %.1f (mm) '
  268 = 'M Enable'
  863 = 'Max %.1f (mm) '
  167 = 'Min %.1f (mm) '
  39 = 'mm'
  116 = 'Mot. Napon(A) %.1f '
  46 = 'Mot. Napon(A) %.3f '
  632 = 'Mot. Napon(V) %.1f '
  265 = 'Mot. Struje(A) %.3f '
  288 = 'Mot.(RPM) %.0f '
  321 = 'Mot.(RPM) %.1f '
  716 = 'MOTOR 1'
  567 = 'MOTOR 2'
  878 = 'MOVE ENABLE'
  703 = 'Moving Neg'
  80 = 'Moving Pos'
  361 = 'Napon M(V) %.1f '
  370 = 'Pozicija %.1f '
  104 = 'Ready '
  115 = 'Ready to EN'
  479 = 'RESET'
  309 = 'Set max Perc %.1f '
  784 = 'Set min Perc %.1f '
  360 = 'Set min Perc %f '
  469 = 'Set Poz %.1f '
  55 = 'Set Vel Perc %.1f '
  343 = 'Sync.Error'
  661 = 'Torq.reduced'
  779 = 'Vel.Overange Neg'
  409 = 'Vel.Overange Poz'
  809 = 'Warning'
END_TEXTLIST

// ---- VISUs/Visualization1.TcVIS
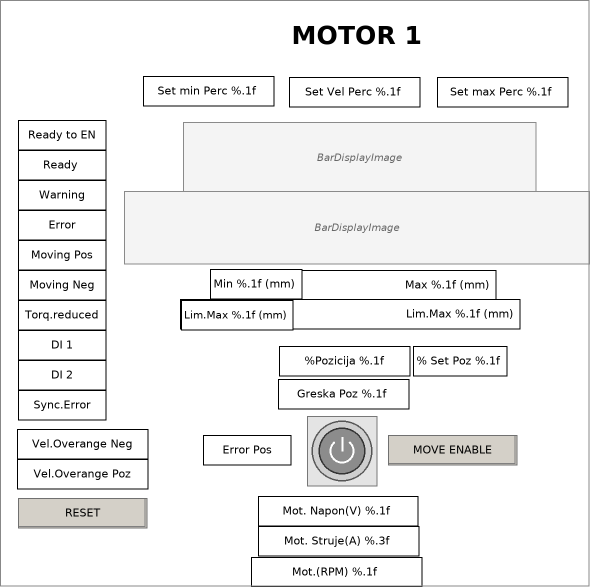
VISUALIZATION Visualization1  // 590x587
    Rectangle (210,270 286x30), "Max %.1f (mm)", text variable: MAIN.FB_DC_MOTOR1.rRadno_Max_Pos
        OnMouseDown: write the text variable via Default, min 0, max 100
    PowerSwitch (307,416 70x70), variable: PRG_ZF_Control.bMotorOn_M1, behaviour: TOGGLE, style: Switch-PowerSwitch-Gray
    Rectangle (143,76 131x30), "Set min Perc %.1f", text variable: MAIN.rSetpointTarget_MinM1
        OnMouseDown: write the text variable via Default, min 0, max 100
    Rectangle (437,77 131x30), "Set max Perc %.1f", text variable: MAIN.rSetpointTarget_MaxM1
        OnMouseDown: write the text variable via Default, min 0, max 100
    Rectangle (279,346 131x30), "%Pozicija %.1f", text variable: MAIN.rPotFeedback_Radno_PercM1
    Rectangle (289,77 131x30), "Set Vel Perc %.1f", text variable: MAIN.rMaxVelocityM1
        OnMouseDown: write the text variable via Default, min 0, max 120
    Rectangle (278,379 131x30), "Greska Poz %.1f", text variable: MAIN.rErrorM1, colour toggle: MAIN.bInDeadband_M1
    Rectangle (258,496 160x30), "Mot. Napon(V) %.1f", text variable: MAIN.rMotorVoltageM1
    Rectangle (258,526 161x30), "Mot. Struje(A) %.3f", text variable: MAIN.rMotorCurrentM1
    Rectangle (413,346 94x30), "% Set Poz %.1f", text variable: MAIN.rSetpointTarget_M1
        OnMouseDown: write the text variable via Default, min 0, max 100
    Rectangle (251,557 171x30), "Mot.(RPM) %.1f", text variable: MAIN.rActualVelocityRPM_M1
    Rectangle (17,429 131x30), "Vel.Overange Neg", colour toggle: MAIN.FB_DC_MOTOR1.bSetVelOverNeg
    Rectangle (17,459 131x30), "Vel.Overange Poz", colour toggle: MAIN.FB_DC_MOTOR1.bSetVelOverPoz
    Button (18,498 129x30), "RESET"
        tap MAIN.bHMI_RESET_M1
    Rectangle (18,120 88x30), "Ready to EN", colour toggle: bReadyToEnable_M1
    Rectangle (18,150 88x30), "Ready", colour toggle: bReady_M1
    Rectangle (18,180 88x30), "Warning", colour toggle: bWarning_M1
    Rectangle (18,210 88x30), "Error", colour toggle: bError_M1
    Rectangle (18,240 88x30), "Moving Pos", colour toggle: bMovingPositive_M1
    Rectangle (18,270 88x30), "Moving Neg", colour toggle: bMovingNegative_M1
    Rectangle (18,300 88x30), "Torq.reduced", colour toggle: bTorqueReduced_M1
    Rectangle (18,330 88x30), "DI 1", colour toggle: bDigitalInput1_M1
    Rectangle (18,360 88x30), "DI 2", colour toggle: bDigitalInput2_M1
    Rectangle (18,390 88x30), "Sync.Error", colour toggle: bSyncError_M1
    Button (388,435 129x30), "MOVE ENABLE", colour toggle: MAIN.bMove_M1
        toggle MAIN.bMove_M1
    BarDisplayImage (183,122 353x71), value: PRG_ZF_Control.rPotFeedback_Radno_PercM1, style: BarDisplayImage-Gray, scale format: %.1f, scale 0..100
        p518627256: %
    BarDisplayImage (124,191 466x73), value: PRG_ZF_Control.FB_DC_MOTOR1.rLinearPosition, style: BarDisplayImage-Gray, scale format: %.1f, scale 0..80
        p518627256: mm
    Rectangle (210,269 92x30), "Min %.1f (mm)", text variable: MAIN.FB_DC_MOTOR1.rRadno_Min_Pos
        OnMouseDown: write the text variable via Default, min 0, max 100
    Rectangle (180,299 340x30), "Lim.Max %.1f (mm)", text variable: MAIN.FB_DC_MOTOR1.rLinearPosition_LimMAx, colour toggle: MAIN.bErrorLimitPosMax_M1
        OnMouseDown: write the text variable via Default, min 0, max 100
    Rectangle (181,300 112x30), "Lim.Max %.1f (mm)", text variable: MAIN.FB_DC_MOTOR1.rLinearPosition_LimMin, colour toggle: MAIN.bErrorLimitPosMin_M1
        OnMouseDown: write the text variable via Default, min 0, max 100
    Label (146,20 422x30), "MOTOR 1"
    Rectangle (203,435 88x30), "Error Pos", colour toggle: MAIN.bERROR_POS_M1
END_VISUALIZATION

// ---- VISUs/Visualization2.TcVIS
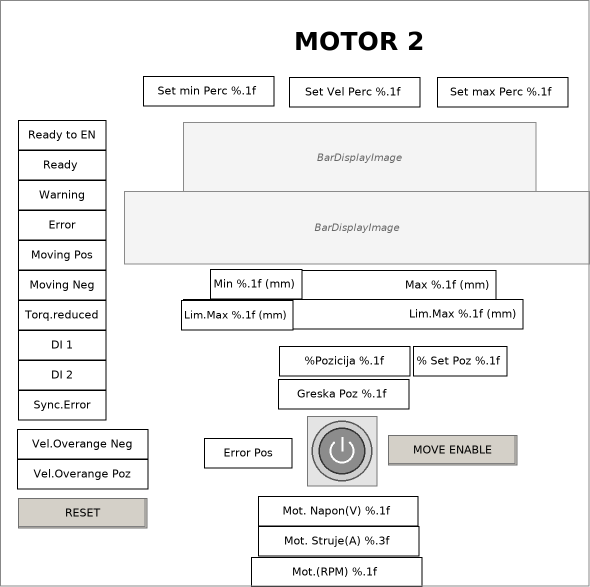
VISUALIZATION Visualization2  // 590x587
    Rectangle (210,270 286x30), "Max %.1f (mm)", text variable: MAIN.FB_DC_MOTOR2.rRadno_Max_Pos
        OnMouseDown: write the text variable via Default, min 0, max 100
    PowerSwitch (307,416 70x70), variable: PRG_ZF_Control.bMotorOn_M2, behaviour: TOGGLE, style: Switch-PowerSwitch-Gray
    Rectangle (143,76 131x30), "Set min Perc %.1f", text variable: MAIN.rSetpointTarget_MinM2
        OnMouseDown: write the text variable via Default, min 0, max 100
    Rectangle (437,77 131x30), "Set max Perc %.1f", text variable: MAIN.rSetpointTarget_MaxM2
        OnMouseDown: write the text variable via Default, min 0, max 100
    Rectangle (279,346 131x30), "%Pozicija %.1f", text variable: MAIN.rPotFeedback_Radno_PercM2
    Rectangle (289,77 131x30), "Set Vel Perc %.1f", text variable: MAIN.rMaxVelocityM2
        OnMouseDown: write the text variable via Default, min 0, max 120
    Rectangle (278,379 131x30), "Greska Poz %.1f", text variable: MAIN.rErrorM2, colour toggle: PRG_ZF_Control.bInDeadband_M2
    Rectangle (258,496 160x30), "Mot. Napon(V) %.1f", text variable: PRG_ZF_Control.rMotorVoltageM2
    Rectangle (258,526 161x30), "Mot. Struje(A) %.3f", text variable: PRG_ZF_Control.rMotorCurrentM2
    Rectangle (413,346 94x30), "% Set Poz %.1f", text variable: MAIN.rSetpointTarget_M2
    Rectangle (251,557 171x30), "Mot.(RPM) %.1f", text variable: PRG_ZF_Control.rActualVelocityRPM_M2
    Rectangle (17,429 131x30), "Vel.Overange Neg", colour toggle: PRG_ZF_Control.FB_DC_MOTOR2.bSetVelOverNeg
    Rectangle (17,459 131x30), "Vel.Overange Poz", colour toggle: PRG_ZF_Control.FB_DC_MOTOR2.bSetVelOverPoz
    Button (18,498 129x30), "RESET"
        tap PRG_ZF_Control.bHMI_RESET_M2
    Rectangle (18,120 88x30), "Ready to EN", colour toggle: bReadyToEnable_M2
    Rectangle (18,150 88x30), "Ready", colour toggle: bReady_M2
    Rectangle (18,180 88x30), "Warning", colour toggle: bWarning_M2
    Rectangle (18,210 88x30), "Error", colour toggle: bError_M2
    Rectangle (18,240 88x30), "Moving Pos", colour toggle: bMovingPositive_M2
    Rectangle (18,270 88x30), "Moving Neg", colour toggle: bMovingNegative_M2
    Rectangle (18,300 88x30), "Torq.reduced", colour toggle: bTorqueReduced_M2
    Rectangle (18,330 88x30), "DI 1", colour toggle: bDigitalInput1_M2
    Rectangle (18,360 88x30), "DI 2", colour toggle: bDigitalInput2_M2
    Rectangle (18,390 88x30), "Sync.Error", colour toggle: bSyncError_M2
    Button (388,435 129x30), "MOVE ENABLE", colour toggle: MAIN.bMove_M2
        toggle PRG_ZF_Control.bMove_M2
    BarDisplayImage (183,122 353x71), value: PRG_ZF_Control.rPotFeedback_Radno_PercM2, style: BarDisplayImage-Gray, scale format: %.1f, scale 0..100
        p518627256: %
    BarDisplayImage (124,191 466x73), value: PRG_ZF_Control.FB_DC_MOTOR2.rLinearPosition, style: BarDisplayImage-Gray, scale format: %.1f, scale 0..80
        p518627256: mm
    Rectangle (210,269 92x30), "Min %.1f (mm)", text variable: MAIN.FB_DC_MOTOR2.rRadno_Min_Pos
        OnMouseDown: write the text variable via Default, min 0, max 100
    Rectangle (183,299 340x30), "Lim.Max %.1f (mm)", text variable: MAIN.FB_DC_MOTOR2.rLinearPosition_LimMAx, colour toggle: MAIN.bErrorLimitPosMax_M2
        OnMouseDown: write the text variable via Default, min 0, max 100
    Rectangle (181,300 112x30), "Lim.Max %.1f (mm)", text variable: MAIN.FB_DC_MOTOR2.rLinearPosition_LimMin, colour toggle: MAIN.bErrorLimitPosMin_M2
        OnMouseDown: write the text variable via Default, min 0, max 100
    Label (148,26 423x30), "MOTOR 2"
    Rectangle (204,438 88x30), "Error Pos", colour toggle: MAIN.bERROR_POS_M2
END_VISUALIZATION

// ---- VISUs/VisuDoorControl.TcVIS
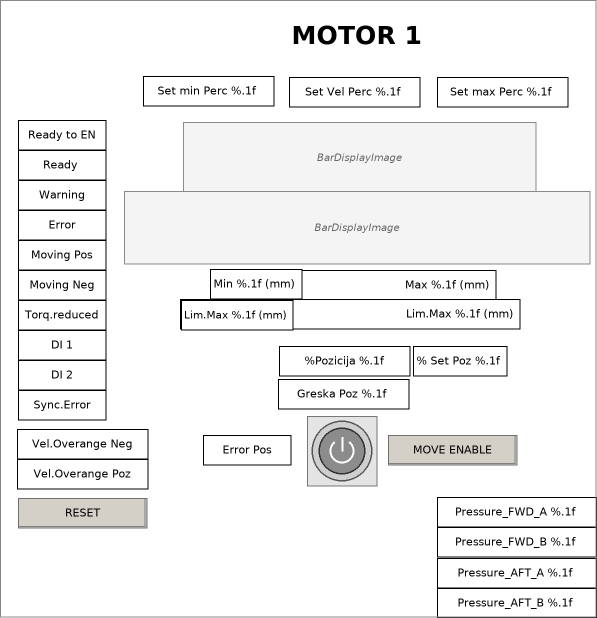
VISUALIZATION VisuDoorControl  // 597x618
    Rectangle (210,270 286x30), "Max %.1f (mm)", text variable: MAIN.FB_DC_MOTOR1.rRadno_Max_Pos
        OnMouseDown: write the text variable via Default, min 0, max 100
    PowerSwitch (307,416 70x70), variable: PRG_ZF_Control.bMotorOn_M1, behaviour: TOGGLE, style: Switch-PowerSwitch-Gray
    Rectangle (143,76 131x30), "Set min Perc %.1f", text variable: MAIN.rSetpointTarget_MinM1
        OnMouseDown: write the text variable via Default, min 0, max 100
    Rectangle (437,77 131x30), "Set max Perc %.1f", text variable: MAIN.rSetpointTarget_MaxM1
        OnMouseDown: write the text variable via Default, min 0, max 100
    Rectangle (279,346 131x30), "%Pozicija %.1f", text variable: MAIN.rPotFeedback_Radno_PercM1
    Rectangle (289,77 131x30), "Set Vel Perc %.1f", text variable: MAIN.rMaxVelocityM1
        OnMouseDown: write the text variable via Default, min 0, max 120
    Rectangle (278,379 131x30), "Greska Poz %.1f", text variable: MAIN.rErrorM1, colour toggle: MAIN.bInDeadband_M1
    Rectangle (413,346 94x30), "% Set Poz %.1f", text variable: MAIN.rSetpointTarget_M1
        OnMouseDown: write the text variable via Default, min 0, max 100
    Rectangle (17,429 131x30), "Vel.Overange Neg", colour toggle: MAIN.FB_DC_MOTOR1.bSetVelOverNeg
    Rectangle (17,459 131x30), "Vel.Overange Poz", colour toggle: MAIN.FB_DC_MOTOR1.bSetVelOverPoz
    Button (18,498 129x30), "RESET"
        tap MAIN.bHMI_RESET_M1
    Rectangle (18,120 88x30), "Ready to EN", colour toggle: bReadyToEnable_M1
    Rectangle (18,150 88x30), "Ready", colour toggle: bReady_M1
    Rectangle (18,180 88x30), "Warning", colour toggle: bWarning_M1
    Rectangle (18,210 88x30), "Error", colour toggle: bError_M1
    Rectangle (18,240 88x30), "Moving Pos", colour toggle: bMovingPositive_M1
    Rectangle (18,270 88x30), "Moving Neg", colour toggle: bMovingNegative_M1
    Rectangle (18,300 88x30), "Torq.reduced", colour toggle: bTorqueReduced_M1
    Rectangle (18,330 88x30), "DI 1", colour toggle: bDigitalInput1_M1
    Rectangle (18,360 88x30), "DI 2", colour toggle: bDigitalInput2_M1
    Rectangle (18,390 88x30), "Sync.Error", colour toggle: bSyncError_M1
    Button (388,435 129x30), "MOVE ENABLE", colour toggle: MAIN.bMove_M1
        toggle MAIN.bMove_M1
    BarDisplayImage (183,122 353x71), value: PRG_ZF_Control.rPotFeedback_Radno_PercM1, style: BarDisplayImage-Gray, scale format: %.1f, scale 0..100
        p518627256: %
    BarDisplayImage (124,191 466x73), value: PRG_ZF_Control.FB_DC_MOTOR1.rLinearPosition, style: BarDisplayImage-Gray, scale format: %.1f, scale 0..80
        p518627256: mm
    Rectangle (210,269 92x30), "Min %.1f (mm)", text variable: MAIN.FB_DC_MOTOR1.rRadno_Min_Pos
        OnMouseDown: write the text variable via Default, min 0, max 100
    Rectangle (180,299 340x30), "Lim.Max %.1f (mm)", text variable: MAIN.FB_DC_MOTOR1.rLinearPosition_LimMAx, colour toggle: MAIN.bErrorLimitPosMax_M1
        OnMouseDown: write the text variable via Default, min 0, max 100
    Rectangle (181,300 112x30), "Lim.Max %.1f (mm)", text variable: MAIN.FB_DC_MOTOR1.rLinearPosition_LimMin, colour toggle: MAIN.bErrorLimitPosMin_M1
        OnMouseDown: write the text variable via Default, min 0, max 100
    Label (146,20 422x30), "MOTOR 1"
    Rectangle (203,435 88x30), "Error Pos", colour toggle: MAIN.bERROR_POS_M1
    Rectangle (437,497 160x30), "Pressure_FWD_A %.1f", text variable: GVL_IO.fPressure_FWD_A
    Rectangle (437,527 160x30), "Pressure_FWD_B %.1f", text variable: GVL_IO.fPressure_FWD_B
    Rectangle (437,558 160x30), "Pressure_AFT_A %.1f", text variable: GVL_IO.fPressure_AFT_A
    Rectangle (437,588 160x30), "Pressure_AFT_B %.1f", text variable: GVL_IO.fPressure_AFT_B
END_VISUALIZATION
